TYPE ST_Axis_InOuts:
STRUCT
// Fizyczne wejścia
	bHomingSensor					AT %I* 	: BOOL;						// Part sensor in Drivesystem 
	wI_DriveInfodata				AT %I* 	: UINT;						// Auxiliary axis data - Digital inputs
	stAxis_Data								: AXIS_REF;					// Main axis data

//Safety Signals
	bQ_SafetyRun AT %Q*: BOOL;
	bQ_SafetyErrorAck AT %Q*: BOOL;
END_STRUCT
END_TYPE

(* stored: Version 1.1.0.1, ProductVersion 3.1.4024.15
   DUT ST_Axis_InOuts: Id {574d86d0-6751-4526-a886-fb667ad466df} *)
